FUNCTION F_LREAL_RoundToPlace : LREAL
VAR_INPUT
    fIn     : LREAL;
    nPlaces : DINT;
END_VAR
VAR
END_VAR

F_LREAL_RoundToPlace := DINT_TO_LREAL(LREAL_TO_DINT(fIn * (nPlaces * 10))) / (nPlaces * 10);

END_FUNCTION

(* stored: Version 1.1.0.1, ProductVersion 3.1.4024.11
   POU F_LREAL_RoundToPlace: Id {637cc13f-6279-4343-aeed-da6cb2a35a31}, SpecialFunc None *)
